(* Logix 5000 project; controller IPG_2332_07A 1769-L16ER-BB1B rev 34.12; software revision 34.01; part 4 of 4 *)
(* tags used below, declared in another part *)
   p_Control : udt_Machine_Control_V2;   // Main Control
   p_FiberAxis : udt_Zaber_Axis;
   p_FiberAxis_FinalMove_Done : BOOL;
   p_FiberAxis_FinalMoveRel : BOOL;
   p_FiberAxis_FindPos : udt_Station_Sequence;
   p_FiberAxis_InitialMove_Done : BOOL;
   p_FiberAxis_InitialMoveRel : BOOL;
   p_FiberAxis_Move_01 : DINT;
   p_FiberAxis_Move_01_String : STRING;
   p_FiberAxis_Move_02 : DINT;
   p_FiberAxis_Move_02_String : STRING;
   p_FiberLength : DINT;
   p_FiberLength_Initial : DINT;
   p_LED_01 : udt_LED;
   p_LED_02 : udt_LED;
   p_LED_03 : udt_LED;
   p_LED_04 : udt_LED;
   p_LED_Ramp : BOOL;
   p_LED_Ramp_Done : BOOL;
(* MainProgram_10Ms, continued *)

ROUTINE L_LED   (* ladder *)
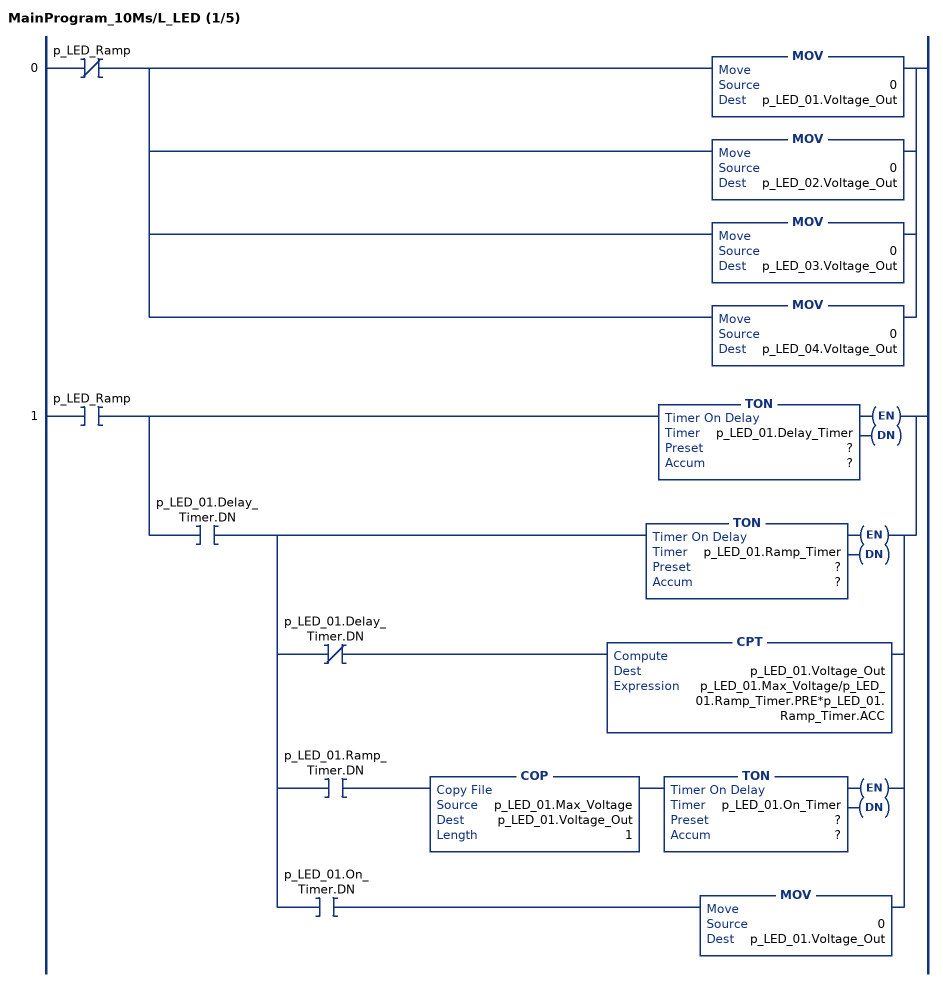
   0: XIO(p_LED_Ramp)[MOV(0,p_LED_01.Voltage_Out) ,MOV(0,p_LED_02.Voltage_Out) ,MOV(0,p_LED_03.Voltage_Out) ,MOV(0,p_LED_04.Voltage_Out) ];
   1: XIC(p_LED_Ramp)[TON(p_LED_01.Delay_Timer,?,?) ,XIC(p_LED_01.Delay_Timer.DN) [TON(p_LED_01.Ramp_Timer,?,?) ,XIO(p_LED_01.Delay_Timer.DN) CPT(p_LED_01.Voltage_Out,p_LED_01.Max_Voltage/p_LED_01.Ramp_Timer.PRE*p_LED_01.Ramp_Timer.ACC) ,XIC(p_LED_01.Ramp_Timer.DN) COP(p_LED_01.Max_Voltage,p_LED_01.Voltage_Out,1) TON(p_LED_01.On_Timer,?,?) ,XIC(p_LED_01.On_Timer.DN) MOV(0,p_LED_01.Voltage_Out) ] ];
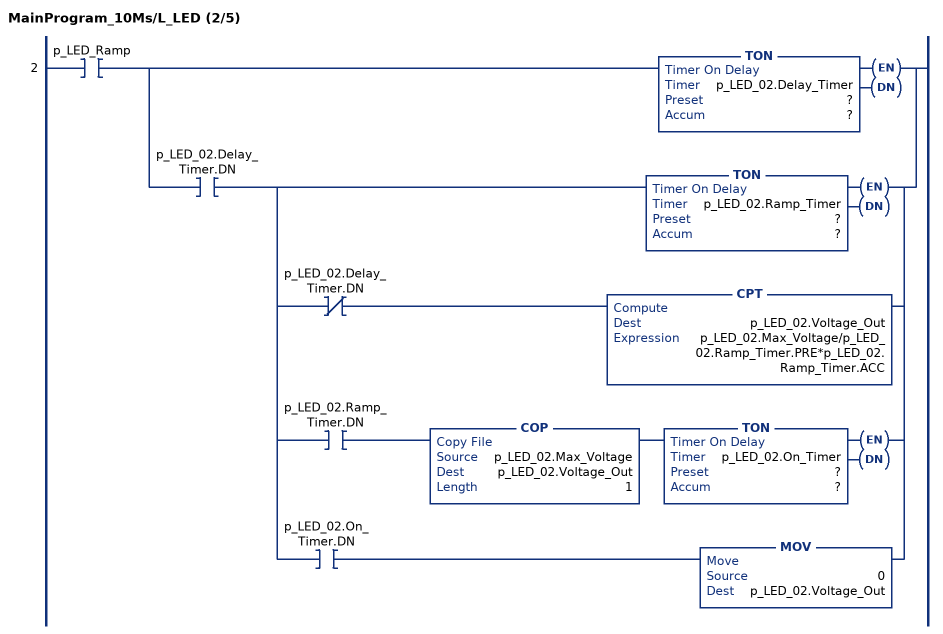
   2: XIC(p_LED_Ramp)[TON(p_LED_02.Delay_Timer,?,?) ,XIC(p_LED_02.Delay_Timer.DN) [TON(p_LED_02.Ramp_Timer,?,?) ,XIO(p_LED_02.Delay_Timer.DN) CPT(p_LED_02.Voltage_Out,p_LED_02.Max_Voltage/p_LED_02.Ramp_Timer.PRE*p_LED_02.Ramp_Timer.ACC) ,XIC(p_LED_02.Ramp_Timer.DN) COP(p_LED_02.Max_Voltage,p_LED_02.Voltage_Out,1) TON(p_LED_02.On_Timer,?,?) ,XIC(p_LED_02.On_Timer.DN) MOV(0,p_LED_02.Voltage_Out) ] ];
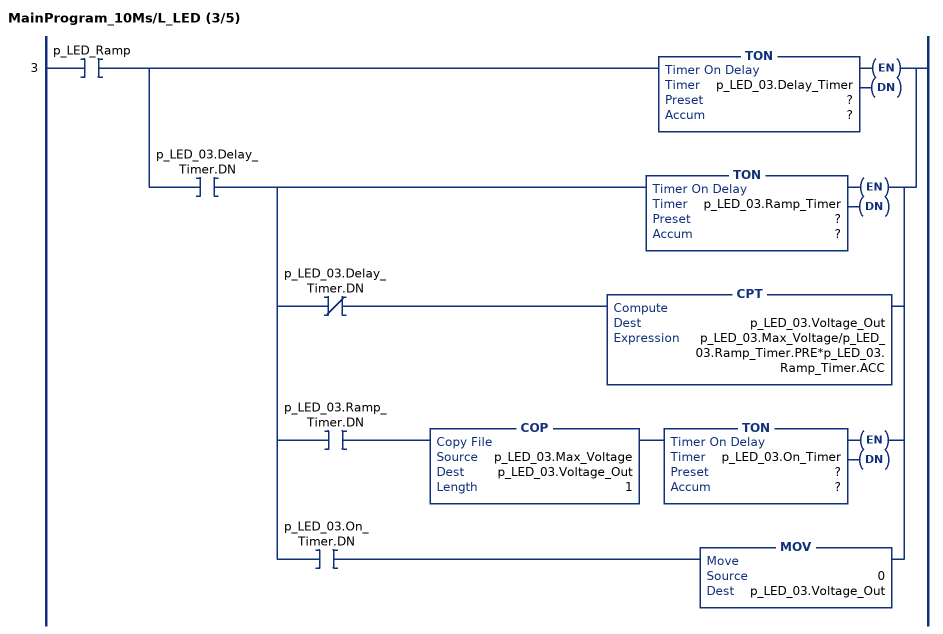
   3: XIC(p_LED_Ramp)[TON(p_LED_03.Delay_Timer,?,?) ,XIC(p_LED_03.Delay_Timer.DN) [TON(p_LED_03.Ramp_Timer,?,?) ,XIO(p_LED_03.Delay_Timer.DN) CPT(p_LED_03.Voltage_Out,p_LED_03.Max_Voltage/p_LED_03.Ramp_Timer.PRE*p_LED_03.Ramp_Timer.ACC) ,XIC(p_LED_03.Ramp_Timer.DN) COP(p_LED_03.Max_Voltage,p_LED_03.Voltage_Out,1) TON(p_LED_03.On_Timer,?,?) ,XIC(p_LED_03.On_Timer.DN) MOV(0,p_LED_03.Voltage_Out) ] ];
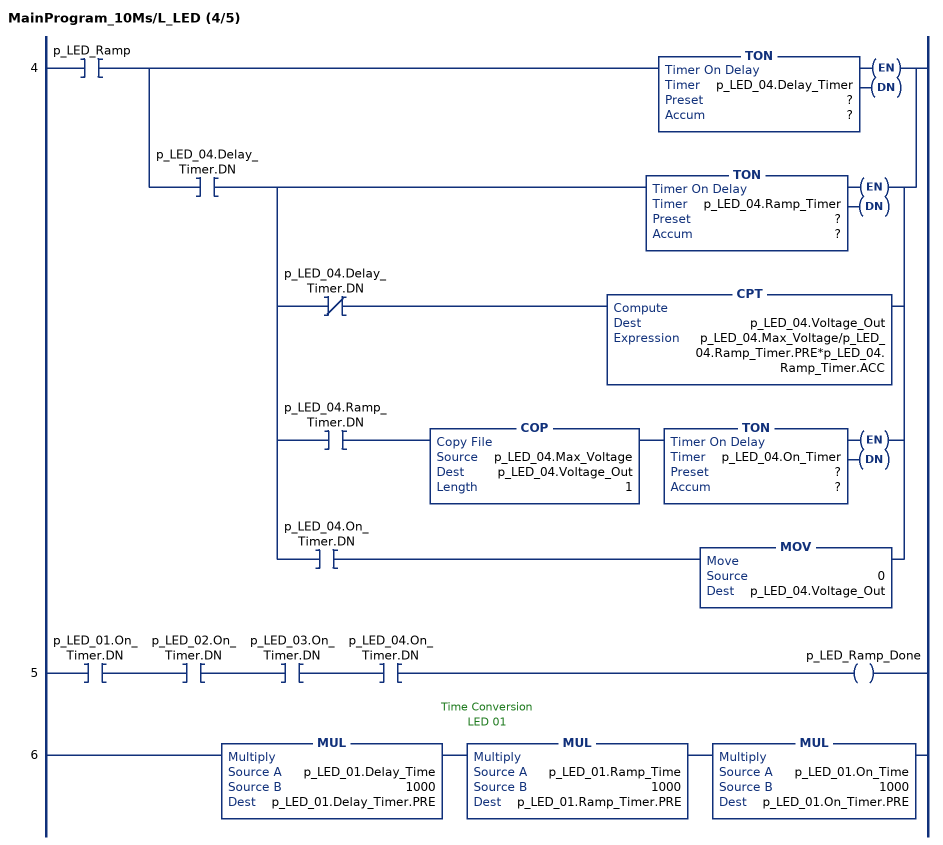
   4: XIC(p_LED_Ramp)[TON(p_LED_04.Delay_Timer,?,?) ,XIC(p_LED_04.Delay_Timer.DN) [TON(p_LED_04.Ramp_Timer,?,?) ,XIO(p_LED_04.Delay_Timer.DN) CPT(p_LED_04.Voltage_Out,p_LED_04.Max_Voltage/p_LED_04.Ramp_Timer.PRE*p_LED_04.Ramp_Timer.ACC) ,XIC(p_LED_04.Ramp_Timer.DN) COP(p_LED_04.Max_Voltage,p_LED_04.Voltage_Out,1) TON(p_LED_04.On_Timer,?,?) ,XIC(p_LED_04.On_Timer.DN) MOV(0,p_LED_04.Voltage_Out) ] ];
   5: XIC(p_LED_01.On_Timer.DN)XIC(p_LED_02.On_Timer.DN)XIC(p_LED_03.On_Timer.DN)XIC(p_LED_04.On_Timer.DN)OTE(p_LED_Ramp_Done);
   // Time Conversion
   // LED 01
   6: MUL(p_LED_01.Delay_Time,1000,p_LED_01.Delay_Timer.PRE)MUL(p_LED_01.Ramp_Time,1000,p_LED_01.Ramp_Timer.PRE)MUL(p_LED_01.On_Time,1000,p_LED_01.On_Timer.PRE);
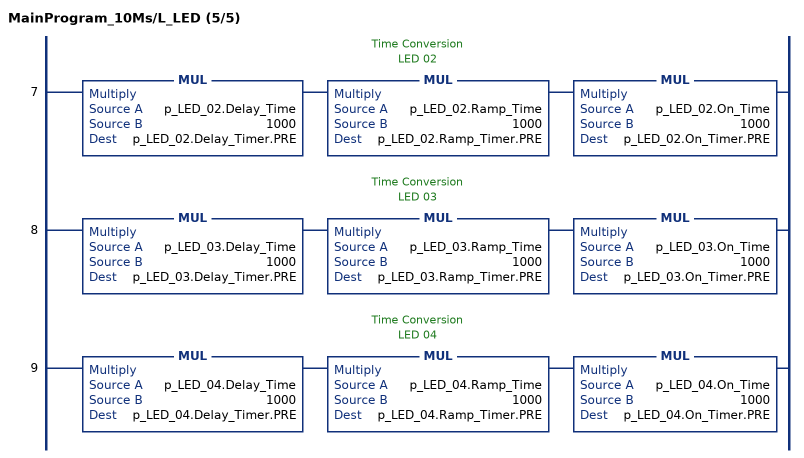
   // Time Conversion
   // LED 02
   7: MUL(p_LED_02.Delay_Time,1000,p_LED_02.Delay_Timer.PRE)MUL(p_LED_02.Ramp_Time,1000,p_LED_02.Ramp_Timer.PRE)MUL(p_LED_02.On_Time,1000,p_LED_02.On_Timer.PRE);
   // Time Conversion
   // LED 03
   8: MUL(p_LED_03.Delay_Time,1000,p_LED_03.Delay_Timer.PRE)MUL(p_LED_03.Ramp_Time,1000,p_LED_03.Ramp_Timer.PRE)MUL(p_LED_03.On_Time,1000,p_LED_03.On_Timer.PRE);
   // Time Conversion
   // LED 04
   9: MUL(p_LED_04.Delay_Time,1000,p_LED_04.Delay_Timer.PRE)MUL(p_LED_04.Ramp_Time,1000,p_LED_04.Ramp_Timer.PRE)MUL(p_LED_04.On_Time,1000,p_LED_04.On_Timer.PRE);
END_ROUTINE

ROUTINE M_FiberAxis_FindPos   (* ladder *)
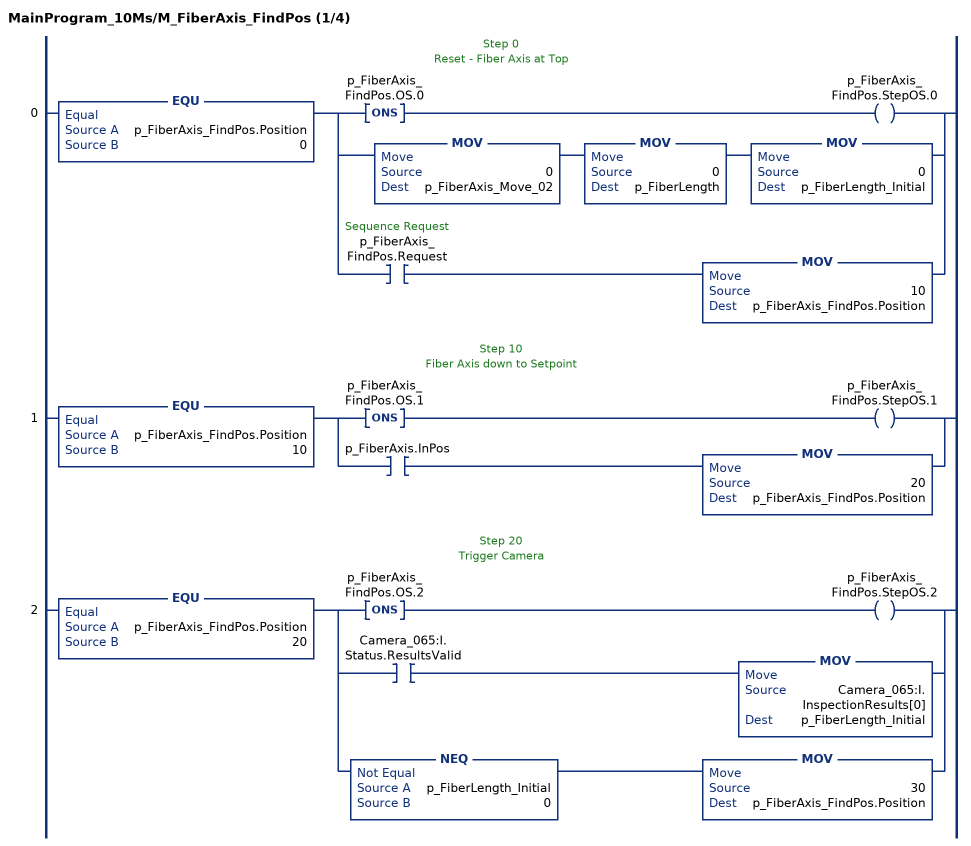
   // Step 0
   // Reset - Fiber Axis at Top
   0: EQU(p_FiberAxis_FindPos.Position,0)[ONS(p_FiberAxis_FindPos.OS.0) OTE(p_FiberAxis_FindPos.StepOS.0) ,MOV(0,p_FiberAxis_Move_02) MOV(0,p_FiberLength) MOV(0,p_FiberLength_Initial) ,XIC(p_FiberAxis_FindPos.Request) MOV(10,p_FiberAxis_FindPos.Position) ];
   // Step 10
   // Fiber Axis down to Setpoint
   1: EQU(p_FiberAxis_FindPos.Position,10)[ONS(p_FiberAxis_FindPos.OS.1) OTE(p_FiberAxis_FindPos.StepOS.1) ,XIC(p_FiberAxis.InPos) MOV(20,p_FiberAxis_FindPos.Position) ];
   // Step 20
   // Trigger Camera
   2: EQU(p_FiberAxis_FindPos.Position,20)[ONS(p_FiberAxis_FindPos.OS.2) OTE(p_FiberAxis_FindPos.StepOS.2) ,XIC(Camera_065:I.Status.ResultsValid) MOV(Camera_065:I.InspectionResults[0],p_FiberLength_Initial) ,NEQ(p_FiberLength_Initial,0) MOV(30,p_FiberAxis_FindPos.Position) ];
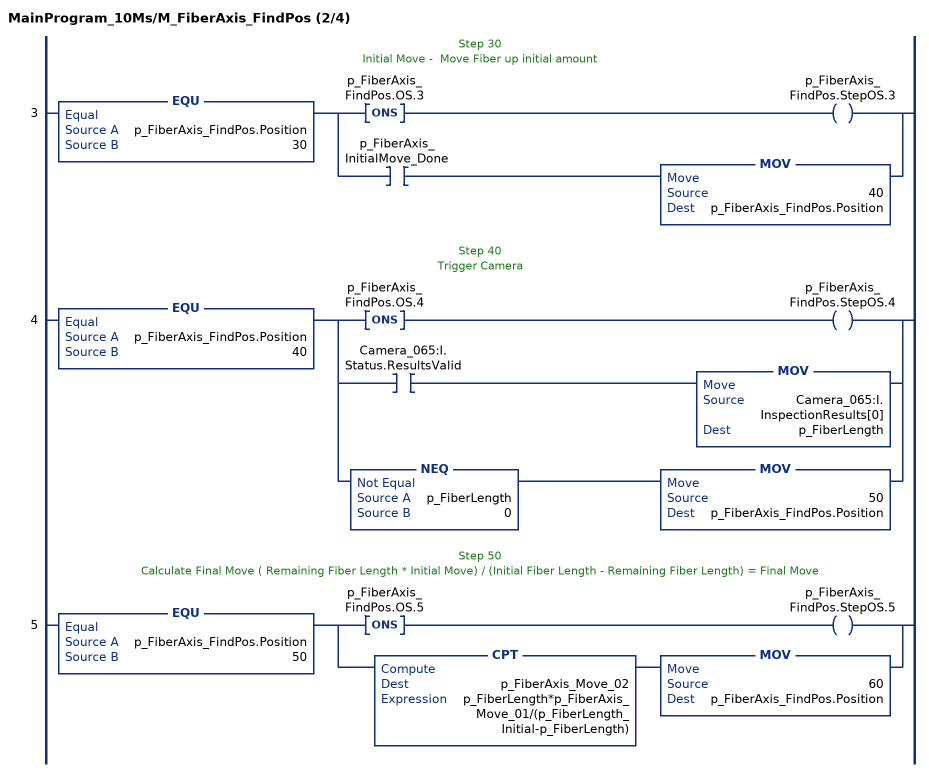
   // Step 30
   // Initial Move -  Move Fiber up initial amount
   3: EQU(p_FiberAxis_FindPos.Position,30)[ONS(p_FiberAxis_FindPos.OS.3) OTE(p_FiberAxis_FindPos.StepOS.3) ,XIC(p_FiberAxis_InitialMove_Done) MOV(40,p_FiberAxis_FindPos.Position) ];
   // Step 40
   // Trigger Camera
   4: EQU(p_FiberAxis_FindPos.Position,40)[ONS(p_FiberAxis_FindPos.OS.4) OTE(p_FiberAxis_FindPos.StepOS.4) ,XIC(Camera_065:I.Status.ResultsValid) MOV(Camera_065:I.InspectionResults[0],p_FiberLength) ,NEQ(p_FiberLength,0) MOV(50,p_FiberAxis_FindPos.Position) ];
   // Step 50
   // Calculate Final Move ( Remaining Fiber Length * Initial Move) / (Initial Fiber Length - Remaining Fiber Length) = Final Move
   5: EQU(p_FiberAxis_FindPos.Position,50)[ONS(p_FiberAxis_FindPos.OS.5) OTE(p_FiberAxis_FindPos.StepOS.5) ,CPT(p_FiberAxis_Move_02,p_FiberLength*p_FiberAxis_Move_01/(p_FiberLength_Initial-p_FiberLength)) MOV(60,p_FiberAxis_FindPos.Position) ];
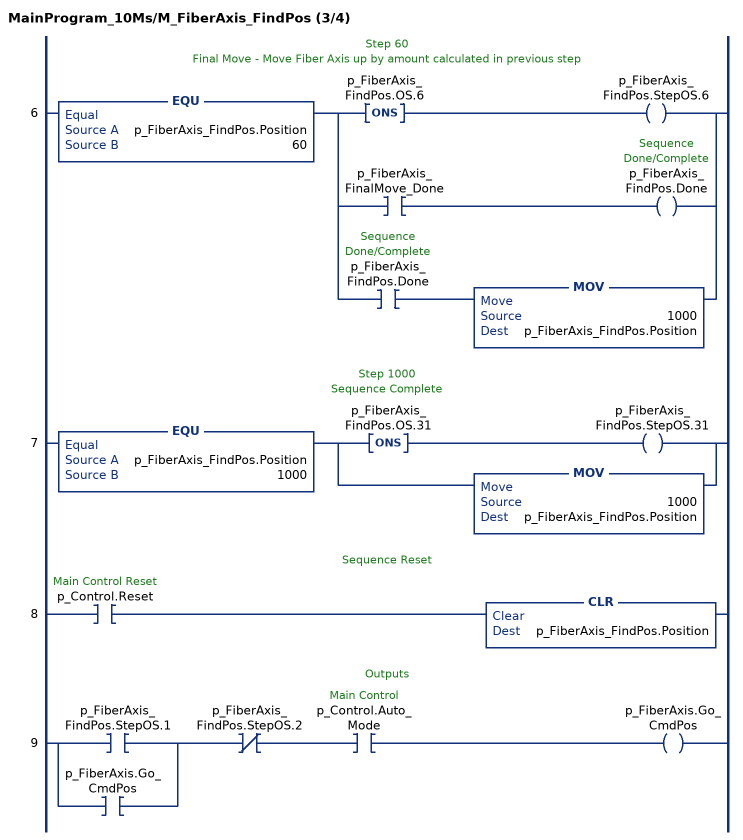
   // Step 60
   // Final Move - Move Fiber Axis up by amount calculated in previous step
   6: EQU(p_FiberAxis_FindPos.Position,60)[ONS(p_FiberAxis_FindPos.OS.6) OTE(p_FiberAxis_FindPos.StepOS.6) ,XIC(p_FiberAxis_FinalMove_Done) OTE(p_FiberAxis_FindPos.Done) ,XIC(p_FiberAxis_FindPos.Done) MOV(1000,p_FiberAxis_FindPos.Position) ];
   // Step 1000
   // Sequence Complete
   7: EQU(p_FiberAxis_FindPos.Position,1000)[ONS(p_FiberAxis_FindPos.OS.31) OTE(p_FiberAxis_FindPos.StepOS.31) ,MOV(1000,p_FiberAxis_FindPos.Position) ];
   // Sequence Reset
   8: XIC(p_Control.Reset)CLR(p_FiberAxis_FindPos.Position);
   // Outputs
   9: [XIC(p_FiberAxis_FindPos.StepOS.1) ,XIC(p_FiberAxis.Go_CmdPos) ]XIO(p_FiberAxis_FindPos.StepOS.2)XIC(p_Control.Auto_Mode)OTE(p_FiberAxis.Go_CmdPos);
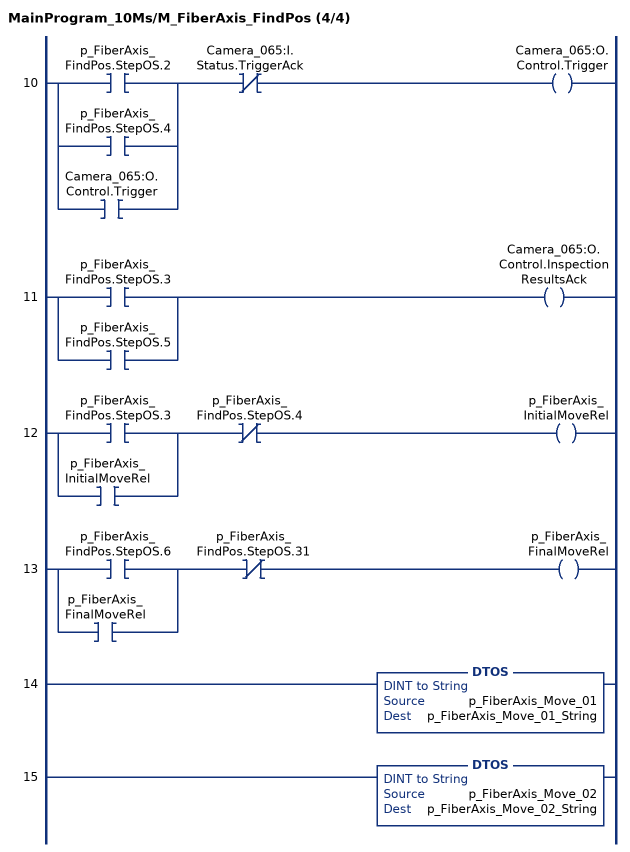
   10: [XIC(p_FiberAxis_FindPos.StepOS.2) ,XIC(p_FiberAxis_FindPos.StepOS.4) ,XIC(Camera_065:O.Control.Trigger) ]XIO(Camera_065:I.Status.TriggerAck)OTE(Camera_065:O.Control.Trigger);
   11: [XIC(p_FiberAxis_FindPos.StepOS.3) ,XIC(p_FiberAxis_FindPos.StepOS.5) ]OTE(Camera_065:O.Control.InspectionResultsAck);
   12: [XIC(p_FiberAxis_FindPos.StepOS.3) ,XIC(p_FiberAxis_InitialMoveRel) ]XIO(p_FiberAxis_FindPos.StepOS.4)OTE(p_FiberAxis_InitialMoveRel);
   13: [XIC(p_FiberAxis_FindPos.StepOS.6) ,XIC(p_FiberAxis_FinalMoveRel) ]XIO(p_FiberAxis_FindPos.StepOS.31)OTE(p_FiberAxis_FinalMoveRel);
   14: DTOS(p_FiberAxis_Move_01,p_FiberAxis_Move_01_String);
   15: DTOS(p_FiberAxis_Move_02,p_FiberAxis_Move_02_String);
END_ROUTINE
END_PROGRAM
